Yaskawa INFORM job: TWIN_FRONT_WELD_90ST-1_5340.JBI

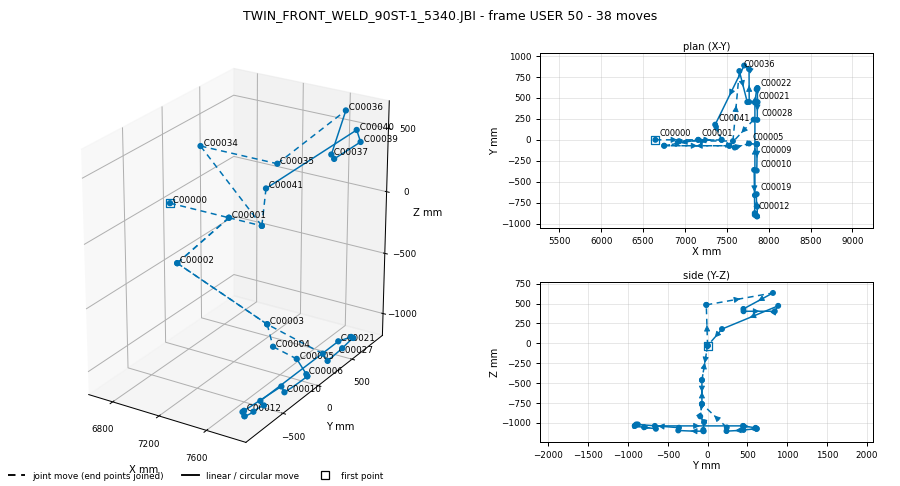
[picture p0: tool path of TWIN_FRONT_WELD_90ST-1_5340.JBI in frame USER 50, 38 of 43 moves have a stored position in this frame; points joined in program order, loops and branches not executed]
/JOB
//NAME TWIN_FRONT_WELD_90ST-1_5340
///FOLDERNAME 02-SKRZYNIE_JOBS
//POS
///NPOS 43,43,0,8,0,0
///USER 50
///TOOL 0
///POSTYPE USER
///RECTAN
///RCONF 0,0,1,0,0,0,0,0,0,0,0,0,0,0,0,0,0,0,0,0,0,0,0,0
C00000=6646.690,0.310,-30.028,0.0000,-53.6567,0.0000
C00001=7158.107,0.308,-30.113,-0.0036,-53.6521,0.0034
///RCONF 1,0,1,0,0,0,0,0,0,0,0,0,0,0,0,0,0,0,0,0,0,0,0,0
C00002=6751.265,-70.527,-461.611,-1.9967,40.9431,160.5509
///RCONF 1,0,0,0,0,0,0,0,0,0,0,0,0,0,0,0,0,0,0,0,0,0,0,0
C00003=7529.702,-70.525,-761.129,-0.1694,36.7808,161.6994
C00004=7593.570,-91.754,-917.210,9.7230,35.0705,163.2693
C00005=7765.780,-43.826,-990.728,-2.4332,41.3600,160.2788
C00006=7853.899,-53.425,-1087.315,-2.4326,41.3464,160.2685
C00007=7860.461,-50.880,-1103.423,-2.4225,41.3460,160.2845
C00008=7860.461,-50.880,-1103.423,-2.4225,41.3460,160.2845
///RCONF 0,0,0,0,0,0,0,0,0,0,0,0,0,0,0,0,0,0,0,0,0,0,0,0
C00009=7860.333,-195.987,-1101.475,-2.5147,41.7064,160.1913
C00010=7856.960,-367.696,-1093.872,-2.5270,41.6997,160.1768
C00011=7825.768,-358.944,-1059.416,-2.5279,41.7009,160.1704
C00012=7833.367,-875.981,-1018.685,38.7242,34.9449,-155.3512
C00013=7833.370,-896.318,-1018.671,38.7251,34.9458,-155.3529
C00014=7860.835,-913.778,-1036.298,38.7246,34.9450,-155.3495
C00015=7860.511,-913.791,-1036.307,38.7248,34.9439,-155.3490
C00016=7862.826,-869.411,-1045.005,33.2123,31.0072,-153.2263
C00017=7861.854,-797.879,-1053.634,32.5926,29.1569,-153.4832
C00018=7854.043,-734.104,-1062.073,32.5803,29.1237,-153.4907
C00019=7856.667,-648.884,-1073.127,32.5651,29.0775,-153.4927
C00020=7835.302,-661.657,-1036.935,32.5695,29.0775,-153.4943
C00021=7835.137,445.512,-1036.569,-41.9938,34.9165,143.3319
C00022=7855.433,603.354,-1061.147,-41.9908,34.9166,143.3377
C00023=7864.649,618.072,-1073.007,-41.9888,34.9189,143.3419
C00024=7864.649,618.067,-1073.010,-41.9885,34.9184,143.3412
///RCONF 0,0,0,0,1,0,0,0,0,0,0,0,0,0,0,0,0,0,0,0,0,0,0,0
C00025=7865.141,526.663,-1080.895,-34.1617,28.5351,130.4088
C00026=7867.301,450.984,-1087.907,-32.0458,27.6493,116.3995
///RCONF 0,0,0,0,0,0,0,0,0,0,0,0,0,0,0,0,0,0,0,0,0,0,0,0
C00027=7864.501,365.563,-1095.054,-32.0403,27.6411,116.4028
C00028=7863.956,238.173,-1102.035,-35.4348,29.0680,114.7796
C00029=7820.420,241.654,-1056.226,-35.4344,29.0737,114.7919
///RCONF 1,0,0,0,0,0,0,0,0,0,0,0,0,0,0,0,0,0,0,0,0,0,0,0
C00030=7529.702,-70.525,-761.129,-0.1694,36.7808,161.6994
///RCONF 1,0,1,0,0,0,0,0,0,0,0,0,0,0,0,0,0,0,0,0,0,0,0,0
C00031=6751.265,-70.527,-461.611,-1.9967,40.9431,160.5509
///RCONF 0,0,1,0,0,0,0,0,0,0,0,0,0,0,0,0,0,0,0,0,0,0,0,0
C00032=7158.107,0.308,-30.113,-0.0036,-53.6521,0.0034
C00033=7437.393,0.308,-30.113,-0.0036,-53.6521,0.0034
///RCONF 1,0,1,0,0,0,0,0,0,0,0,0,0,0,0,0,0,0,0,0,0,0,0,0
C00034=6928.400,-15.669,483.666,2.7707,-42.5282,-1.8493
C00035=7572.625,-15.669,483.666,2.7707,-42.5282,-1.8493
C00036=7649.331,821.904,633.544,31.3308,-50.3097,5.8371
C00037=7744.044,450.716,432.605,31.3340,-50.3098,5.8344
C00038=7767.030,452.216,403.290,-5.2996,-47.7530,32.0852
C00039=7765.112,844.716,403.608,27.6981,-50.7461,8.3527
C00040=7706.752,887.668,471.666,31.3375,-50.3103,5.8310
C00041=7360.642,181.544,179.903,-30.3084,-22.7119,47.7634
///RCONF 0,0,1,0,0,0,0,0,0,0,0,0,0,0,0,0,0,0,0,0,0,0,0,0
C00042=7437.393,0.308,-30.113,-0.0036,-53.6521,0.0034
///RCONF 0,0,0,0,0,0,0,0,0,0,0,0,0,0,0,0,0,0,0,0,0,0,0,0
BC00000=4832.263
BC00001=5343.689
BC00002=5343.689
BC00003=6178.800
BC00004=6423.804
BC00005=6624.475
BC00006=6624.475
BC00007=6624.482
BC00008=6624.482
BC00009=6624.488
BC00010=6624.482
BC00011=6624.482
BC00012=6624.488
BC00013=6624.488
BC00014=6624.488
BC00015=6624.488
BC00016=6624.489
BC00017=6624.879
BC00018=6624.710
BC00019=6624.489
BC00020=6624.488
BC00021=6624.488
BC00022=6624.482
BC00023=6624.482
BC00024=6624.482
BC00025=6624.482
BC00026=6624.482
BC00027=6624.482
BC00028=6624.482
BC00029=6624.482
BC00030=6178.800
BC00031=5343.689
BC00032=5343.689
BC00033=5622.975
BC00034=5622.975
BC00035=6267.199
BC00036=6480.663
BC00037=6480.663
BC00038=6480.663
BC00039=6480.644
BC00040=6480.663
BC00041=6140.736
BC00042=5622.975
///POSTYPE BASE
P00021=6.550,-0.003,-5.735,0.0000,0.0000,0.0000
P00022=5.943,-0.018,-6.388,0.0000,0.0000,0.0000
///RCONF 1,0,0,0,0,0,0,0,0,0,0,0,0,0,0,0,0,0,0,0,0,0,0,0
P00500=2.332,-5.281,-1.258,0.0000,0.0000,0.0000
///RCONF 0,0,0,0,0,0,0,0,0,0,0,0,0,0,0,0,0,0,0,0,0,0,0,0
P00501=-2.026,0.009,3.534,0.0000,0.0000,0.0000
///RCONF 1,0,0,0,0,0,0,0,0,0,0,0,0,0,0,0,0,0,0,0,0,0,0,0
P00502=-2.023,0.001,1.732,0.0000,0.0000,0.0000
P00503=0.138,-0.044,1.539,0.0000,0.0000,0.0000
P00504=-0.309,-0.010,1.636,0.0000,0.0000,0.0000
P00505=0.999,-9.916,8.214,0.0000,0.0000,0.0000
//INST
///DATE 2024/12/18 12:50
///ATTR SC,RW,RJ
////FRAME USER 50
///GROUP1 RB1,BS1
NOP
MOVJ C00000 BC00000 VJ=80.00
MOVJ C00001 BC00001 VJ=50.00
MOVJ C00002 BC00002 VJ=50.00
MOVJ C00003 BC00003 VJ=50.00
MOVJ C00004 BC00004 VJ=50.00
MOVJ C00005 BC00005 VJ=30.00
'::::::::::::::::::::::::::::::::
'W20
'::::::::::::::::::::::::::::::::
MOVL C00006 BC00006 V=333.3
SFTON P0503
MACRO1 MJ#(0) ARGF14
MOVL C00007 BC00007 V=133.3 PL=0
ARCON
MOVC C00008 BC00008 V=9.5
MOVC C00009 BC00009 V=9.5
SFTOF
SFTON P0502
MOVC C00010 BC00010 V=9.5
ARCOF
MOVL C00011 BC00011 V=250.0
SFTOF
MOVL C00012 BC00012 V=250.0
'::::::::::::::::::::::::::::::::
'W21
'::::::::::::::::::::::::::::::::
MOVL C00013 BC00013 V=166.7
SFTON P0500
MACRO1 MJ#(0) ARGF14
MOVL C00014 BC00014 V=133.3 PL=0
ARCON
MOVC C00015 BC00015 V=9.5
MOVC C00016 BC00016 V=9.5
MOVC C00017 BC00017 V=9.5
SFTOF
SFTON P0501
MOVC C00018 BC00018 V=9.5
MOVC C00019 BC00019 V=9.5
ARCOF
MOVL C00020 BC00020 V=250.0
SFTOF
MOVL C00021 BC00021 V=333.3
'::::::::::::::::::::::::::::::::
'W22
'::::::::::::::::::::::::::::::::
MOVL C00022 BC00022 V=166.7
SFTON P0505
MACRO1 MJ#(0) ARGF14
MOVL C00023 BC00023 V=133.3 PL=0
ARCON
MOVC C00024 BC00024 V=9.5
MOVC C00025 BC00025 V=9.5
MOVC C00026 BC00026 V=9.5
SFTOF
SFTON P0504
MOVC C00027 BC00027 V=9.5
MOVC C00028 BC00028 V=9.5
ARCOF
MOVL C00029 BC00029 V=166.7
SFTOF
MOVJ C00030 BC00030 VJ=50.00
MOVJ C00031 BC00031 VJ=80.00
MOVJ C00032 BC00032 VJ=80.00
MOVJ C00033 BC00033 VJ=50.00
MOVJ C00034 BC00034 VJ=50.00
MOVJ C00035 BC00035 VJ=50.00
MOVJ C00036 BC00036 VJ=50.00
MOVL C00037 BC00037 V=166.7
PAUSE
'SPRAWDZIC
SFTON P0022
MOVL C00038 BC00038 V=166.7
ARCON
SFTON P0021
MOVL C00039 BC00039 V=7.5
ARCOF
MOVL C00040 BC00040 V=166.7
SFTOF
MOVL C00041 BC00041 V=333.3
MOVJ C00042 BC00042 VJ=50.00
END
